{attribute 'OPC.UA.DA.StructuredType' := '1'}
{attribute 'OPC.UA.DA' := '1'}
TYPE stExternalStatus :
STRUCT
	SKILLID				: UINT;
	SKILLNAME			: STRING;
	ExecutionBusy		: BOOL;
    ExecutionDone       : BOOL;
	ExecutionResult		: eResult;
END_STRUCT
END_TYPE

(* stored: Version 1.1.0.1, ProductVersion 3.1.4026.18
   DUT stExternalStatus: Id {66db3fe8-3949-42e4-8d15-d5cb7cd19d5b} *)
